{attribute 'enable_dynamic_creation'}
TYPE Struct1 :
STRUCT
	bIn : BOOL;
	iIn : INT;
END_STRUCT
END_TYPE

(* stored: Version 1.1.0.1, ProductVersion 3.1.4024.11
   DUT Struct1: Id {b7deaa78-7cc7-463d-8848-17a34c98d760} *)
